TYPE ST_VisuCtrlCylinderFrame EXTENDS ST_VisuCtrlUnitFrame :
STRUCT
	btnInit				: BOOL;				(*  *)
	btnAbort			: BOOL;				(*  *)
	btnReset			: BOOL;				(*  *)
	btnGoHome 			: BOOL;				(*  *)
	btnGoActive 		: BOOL;				(*  *)
	btnRealase 			: BOOL;				(*  *)
	
	bSensorHome 		: BOOL;				(*  *)
	bSensorActive 		: BOOL;				(*  *)
	bPositionHold		: BOOL;				(*  *)
	bError				: BOOL;				(*  *)
	iErrorID			: INT;				(*  *)
	
	tActiveMovement 	: TIME;				(*  *)
	tHomeMovement 		: TIME;				(*  *)
	
	sActiveDescription 	: STRING;			(*  *)
	sHomeDescription 	: STRING;			(*  *)
	sStateDescription	: STRING;			(*  *)
	
	sCylinderImage		: STRING;			(*  *)
	eCylinderState		: E_CylinderState;	(*  *)
END_STRUCT
END_TYPE

(* stored: Version 1.1.0.1, ProductVersion 3.1.4024.9
   DUT ST_VisuCtrlCylinderFrame: Id {27e27e36-55fd-4b1a-83b6-65bb568807df} *)
